// TIA Portal V19 export
FUNCTION "ERROR_MSG_CLEAR" : Void   // FC218, STL
TITLE = Clear error messages after configured delay
{ S7_Optimized_Access := 'TRUE' }
AUTHOR : HGS
FAMILY : MESSAGES
NAME : CLEAR
// stored: AutoNumber false
   VAR_INPUT
      MESSAGE_CLEAR_TIME : Int;   // Time before clearing message (seconds)
      SECOND_PULSE : Bool;   // second pulse (1Hz)
   END_VAR
   VAR_IN_OUT
      ERROR_MESSAGE : Int;   // Error message to be cleared
      ERROR_MESSAGE_MEM : Int;   // Memory of error message
      ELAPSED_TIME : Int;   // Actual time after message change
   END_VAR
   VAR_TEMP
      ERROR_MESSAGE_CHANGED : Bool;   // Error message has changed
   END_VAR
BEGIN

NETWORK
TITLE = Check if a message is present
      L     #ERROR_MESSAGE;
      L     0;
      ==I;
      BEC;


NETWORK
TITLE = Time the error message
      L     #ERROR_MESSAGE;
      L     #ERROR_MESSAGE_MEM;
      <>I;
      =     #ERROR_MESSAGE_CHANGED;

      L     #ERROR_MESSAGE;
      T     #ERROR_MESSAGE_MEM;

      AN    #ERROR_MESSAGE_CHANGED;
      JC    dL06;

      L     0;
      T     #ELAPSED_TIME;

dL06: NOP   0;


      L     #MESSAGE_CLEAR_TIME;
      L     1;
      *I;
      L     #ELAPSED_TIME;
      >I;
      JC    dL15;

      L     0;
      T     #ERROR_MESSAGE;
      T     #ELAPSED_TIME;
      T     #ERROR_MESSAGE_MEM;

dL15: NOP   0;

      AN    #SECOND_PULSE;
      JC    dL03;

      L     #ELAPSED_TIME;
      L     1;
      +I;
      T     #ELAPSED_TIME;

dL03: NOP   0;
END_FUNCTION
